SUBAPPLICATION SoftKeySRT_ASRT_AX (* 3 SoftKeys (Set/Reset/Toggle) und GreenWhiteBackground am Toggle-SoftKey, gebuendelt hinter einem einzigen ASRT_AX-Plug (bidirektional: Set/Reset/Toggle raus, Zustand rein) - HMI-Teil, ohne jeden OPC-UA-Bezug, wiederverwendbar *)
  (* Standard: 61499-2; Description: Copyright (c) 2026 Meisterschulen am Ostbahnhof This program and the accompanying materials are made available under the terms of the Eclipse Public License 2.0 which is available at https://www.eclipse.org/legal/epl-2.0/ SPDX-License-Identifier: EPL-2.0 *)
  (* Version 1.0, 2026-09-04, Franz Höpfinger, Meisterschulen am Ostbahnhof, initial API and implementation and/or initial documentation *)
  PACKAGE MyLib::sys;
  IMPORT isobus::UT::Q::const::IDs::ID_NULL;
  IMPORT isobus::UT::io::Softkey::SoftKeyActivationCode::SK_RELEASED;
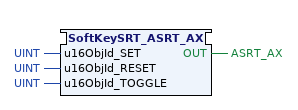
  VAR_INPUT
    u16ObjId_SET : UINT := ID_NULL; (* Object ID SoftKey Set *)
    u16ObjId_RESET : UINT := ID_NULL; (* Object ID SoftKey Reset *)
    u16ObjId_TOGGLE : UINT := ID_NULL; (* Object ID SoftKey Toggle (traegt auch das GreenWhiteBackground) *)
  END_VAR
  PLUGS
    OUT : adapter::types::bidirectional::ASRT_AX; (* Set/Reset/Toggle (out), Zustand (in) *)
  END_PLUGS
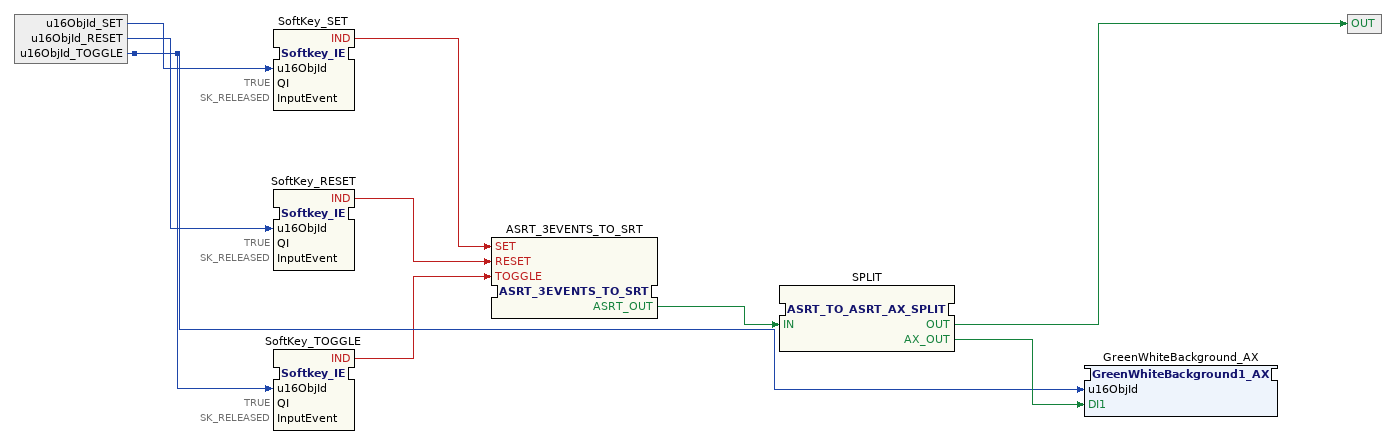
  FBS
    SoftKey_SET : isobus::UT::io::Softkey::Softkey_IE(QI := TRUE, InputEvent := SK_RELEASED);
    SoftKey_RESET : isobus::UT::io::Softkey::Softkey_IE(QI := TRUE, InputEvent := SK_RELEASED);
    SoftKey_TOGGLE : isobus::UT::io::Softkey::Softkey_IE(QI := TRUE, InputEvent := SK_RELEASED);
    SPLIT : adapter::events::bidirectional::ASRT_TO_ASRT_AX_SPLIT;
    ASRT_3EVENTS_TO_SRT : adapter::conversion::unidirectional::ASRT_3EVENTS_TO_SRT;
  END_FBS
  SUBAPPS
    GreenWhiteBackground_AX : MyLib::sys::GreenWhiteBackground1_AX;
  END_SUBAPPS
  EVENT_CONNECTIONS
    SoftKey_SET.IND TO ASRT_3EVENTS_TO_SRT.SET;
    SoftKey_RESET.IND TO ASRT_3EVENTS_TO_SRT.RESET;
    SoftKey_TOGGLE.IND TO ASRT_3EVENTS_TO_SRT.TOGGLE;
  END_CONNECTIONS
  DATA_CONNECTIONS
    u16ObjId_SET TO SoftKey_SET.u16ObjId;
    u16ObjId_RESET TO SoftKey_RESET.u16ObjId;
    u16ObjId_TOGGLE TO SoftKey_TOGGLE.u16ObjId;
    u16ObjId_TOGGLE TO GreenWhiteBackground_AX.u16ObjId;
  END_CONNECTIONS
  ADAPTER_CONNECTIONS
    ASRT_3EVENTS_TO_SRT.ASRT_OUT TO SPLIT.IN;
    SPLIT.OUT TO OUT;
    SPLIT.AX_OUT TO GreenWhiteBackground_AX.DI1;
  END_CONNECTIONS
END_SUBAPPLICATION
